(* IEC 61131-3 sources: ESP32-PLC/openPLC-files/conexiones/build, 2 files *)

(* ---- plc.st ---- *)
TYPE
  LOGLEVEL : (CRITICAL, WARNING, INFO, DEBUG) := INFO;
END_TYPE

FUNCTION_BLOCK LOGGER
  VAR_INPUT
    TRIG : BOOL;
    MSG : STRING;
    LEVEL : LOGLEVEL := INFO;
  END_VAR
  VAR
    TRIG0 : BOOL;
  END_VAR

  IF TRIG AND NOT TRIG0 THEN
  {{
   LogMessage(GetFbVar(LEVEL),(char*)GetFbVar(MSG, .body),GetFbVar(MSG, .len));
  }}
  END_IF;
  TRIG0:=TRIG;
END_FUNCTION_BLOCK

PROGRAM conexiones
  VAR
    TON0 : TON;
    TON1 : TON;
  END_VAR
  VAR
    Pardada AT %IX0.0 : BOOL;
    Conmutar AT %IX0.4 : BOOL;
  END_VAR
  VAR
    Cambiar : BOOL;
    Detener : BOOL;
  END_VAR
  VAR
    Delta AT %QX0.5 : BOOL;
    Estrella AT %QX0.6 : BOOL;
  END_VAR
  VAR
    YOn : BOOL;
    YOnAux : BOOL;
    DosOff : BOOL;
    DosOffAux : BOOL;
    TON2 : TON;
    TON3 : TON;
  END_VAR

  Detener := NOT(Conmutar) AND (Detener OR Pardada);
  TON1(IN := NOT(DosOffAux) AND NOT(DosOff) AND NOT(Cambiar) AND NOT(Detener), PT := T#10000ms);
  YOn := TON1.Q;
  TON0(IN := NOT(DosOff) AND (YOn OR YOnAux) AND NOT(Cambiar) AND NOT(Detener), PT := T#10000ms);
  DosOff := TON0.Q;
  Delta := NOT(YOnAux) AND NOT(YOn) AND NOT(Detener);
  Estrella := (YOn OR YOnAux) AND NOT(Detener);
  TON2(IN := (Cambiar AND NOT(Estrella) OR NOT(DosOffAux) AND NOT(DosOff) AND YOnAux) AND NOT(Detener), PT := T#500ms);
  YOnAux := TON2.Q;
  TON3(IN := Cambiar AND NOT(Delta) AND NOT(Detener), PT := T#500ms);
  DosOffAux := TON3.Q;
  Cambiar := NOT(DosOffAux) AND NOT(DosOff) AND (Cambiar OR NOT(Detener) AND Conmutar);
END_PROGRAM

CONFIGURATION Config0

  RESOURCE Res0 ON PLC
    TASK task0(INTERVAL := T#20ms,PRIORITY := 0);
    PROGRAM instance0 WITH task0 : conexiones;
  END_RESOURCE
END_CONFIGURATION

(* ---- generated_plc.st ---- *)
PROGRAM conexiones
  VAR
    TON0 : TON;
    TON1 : TON;
  END_VAR
  VAR
    Pardada AT %IX0.0 : BOOL;
    Conmutar AT %IX0.4 : BOOL;
  END_VAR
  VAR
    Cambiar : BOOL;
    Detener : BOOL;
  END_VAR
  VAR
    Delta AT %QX0.5 : BOOL;
    Estrella AT %QX0.6 : BOOL;
  END_VAR
  VAR
    YOn : BOOL;
    YOnAux : BOOL;
    DosOff : BOOL;
    DosOffAux : BOOL;
    TON2 : TON;
    TON3 : TON;
  END_VAR

  Detener := NOT(Conmutar) AND (Detener OR Pardada);
  TON1(IN := NOT(DosOffAux) AND NOT(DosOff) AND NOT(Cambiar) AND NOT(Detener), PT := T#10000ms);
  YOn := TON1.Q;
  TON0(IN := NOT(DosOff) AND (YOn OR YOnAux) AND NOT(Cambiar) AND NOT(Detener), PT := T#10000ms);
  DosOff := TON0.Q;
  Delta := NOT(YOnAux) AND NOT(YOn) AND NOT(Detener);
  Estrella := (YOn OR YOnAux) AND NOT(Detener);
  TON2(IN := (Cambiar AND NOT(Estrella) OR NOT(DosOffAux) AND NOT(DosOff) AND YOnAux) AND NOT(Detener), PT := T#500ms);
  YOnAux := TON2.Q;
  TON3(IN := Cambiar AND NOT(Delta) AND NOT(Detener), PT := T#500ms);
  DosOffAux := TON3.Q;
  Cambiar := NOT(DosOffAux) AND NOT(DosOff) AND (Cambiar OR NOT(Detener) AND Conmutar);
END_PROGRAM

CONFIGURATION Config0

  RESOURCE Res0 ON PLC
    TASK task0(INTERVAL := T#20ms,PRIORITY := 0);
    PROGRAM instance0 WITH task0 : conexiones;
  END_RESOURCE
END_CONFIGURATION
